SUBAPPLICATION SoftKey_Kurz_Lang_5s (* Unterscheidet kurzen Tastendruck (Loslassen vor 5s) von langem Tastendruck (5s gehalten) auf einem AX-Adapter-Eingang (z.B. Softkey_IXA.IN). LANG feuert sofort beim Erreichen von 5s (nicht erst beim Loslassen); KURZ feuert beim Loslassen, wenn 5s noch nicht erreicht waren. *)
  (* Standard: 61499-2; Description: Copyright (c) 2026 Meisterschulen am Ostbahnhof This program and the accompanying materials are made available under the terms of the Eclipse Public License 2.0 which is available at https://www.eclipse.org/legal/epl-2.0/ SPDX-License-Identifier: EPL-2.0 *)
  (* Version 1.0, 2026-09-11, Franz Höpfinger, Meisterschulen am Ostbahnhof, initial implementation - fuer Achslenkung-Mittelpunkt-Taste (kurz=Anfahren, lang=Speichern), generisch fuer jede Softkey-Kurz/Lang-Unterscheidung *)
  PACKAGE MyLib::sys;
  (* Documentation:
  Kurz/Lang-Druck-Unterscheidung (5s)
   E_TON (AX_TON, PT=5s) laeuft solange IN gehalten wird. R_TRIG_LONG erkennt die steigende Flanke von E_TON.Q - das ist der Moment, in dem 5s erreicht sind, waehrend die Taste noch gehalten wird - und feuert LANG sofort, ohne auf das Loslassen zu warten.
   F_TRIG_RELEASE erkennt die fallende Flanke von IN (Loslassen). PERMIT_KURZ (AX_E_PERMIT_INVERT_1) laesst dieses Ereignis nur durch, wenn E_TON.Q zu diesem Zeitpunkt noch FALSE ist - also wenn losgelassen wurde, BEVOR 5s erreicht waren. Wurde bereits LANG gefeuert, unterdrueckt PERMIT_KURZ das nachtraegliche KURZ beim Loslassen.
  *)
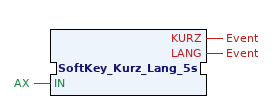
  EVENT_OUTPUT
    KURZ; (* Kurzer Druck bestaetigt (Loslassen vor Ablauf 5s) *)
    LANG; (* Langer Druck bestaetigt (5s erreicht, feuert sofort - nicht erst beim Loslassen) *)
  END_EVENT
  SOCKETS
    IN : adapter::types::unidirectional::AX; (* Rohzustand der Taste (z.B. Softkey_IXA.IN) *)
  END_SOCKETS
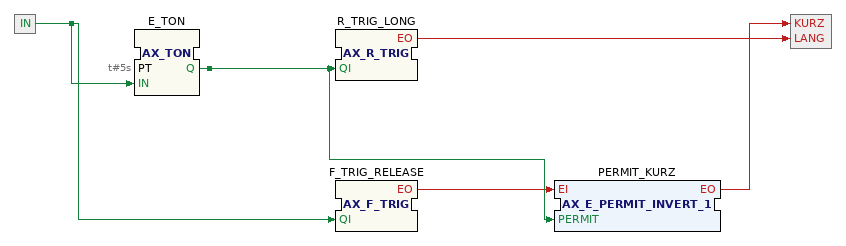
  FBS
    E_TON : adapter::events::unidirectional::timers::AX_TON(PT := t#5s);
    R_TRIG_LONG : adapter::events::unidirectional::AX_R_TRIG;
    F_TRIG_RELEASE : adapter::events::unidirectional::AX_F_TRIG;
  END_FBS
  SUBAPPS
    PERMIT_KURZ : MyLib::sys::AX_E_PERMIT_INVERT_1;
  END_SUBAPPS
  EVENT_CONNECTIONS
    R_TRIG_LONG.EO TO LANG;
    F_TRIG_RELEASE.EO TO PERMIT_KURZ.EI;
    PERMIT_KURZ.EO TO KURZ;
  END_CONNECTIONS
  ADAPTER_CONNECTIONS
    IN TO E_TON.IN;
    IN TO F_TRIG_RELEASE.QI;
    E_TON.Q TO R_TRIG_LONG.QI;
    E_TON.Q TO PERMIT_KURZ.PERMIT;
  END_CONNECTIONS
END_SUBAPPLICATION
